// TIA Portal V20 export
// export: Created 2025-12-01T14:57:08.5701535Z, ExportSetting None, DisplayName Totally Integrated Automation Portal, DisplayVersion V20 Update 3, DisplayName TIA Portal Openness, DisplayVersion V20 Update 3, DisplayName TIA Portal Version Control Interface, DisplayVersion V20 Update 3, DisplayName STEP 7 Professional, DisplayVersion V20 Update 3, DisplayName STEP 7 Safety, DisplayVersion V20 Update 2, DisplayName WinCC Basic/Comfort/Advanced, DisplayVersion V20 Update 3, DisplayName WinCC Professional, DisplayVersion V20 Update 3, DisplayName WinCC Unified, DisplayVersion V20 Update 3
FUNCTION "FC918_GestorAccesos" : Void   // FC918, LAD
{ S7_Optimized_Access := 'FALSE' }
// stored: AutoNumber false, SetENOAutomatically false
   VAR_INPUT
      Numero : UInt;
      ModoPulsador : Bool;
      PermisoActivarPeticion : Bool;
      PermisoDesActivarPeticion : Bool;
      S_Peticion : Bool;
   END_VAR
   VAR_OUTPUT
      H_Permiso : Bool;
      NoEntrarCarga : Bool;
      BloqueoPuerta : Bool;
   END_VAR
   VAR_TEMP
      Acceso : "UDT_Accesos";
      PAny_DB_Acceso : Any;
      Guardar_AR2 : DWord;
      P_ArrayMesas : DWord;
      P_Acceso : DWord;
      ReturnValor : Int;
      Long_Accesos : UInt;
      NDB_Accesos : UInt;
      NMesas_Accesos : UInt;
      Indice : UInt;
      Mesa : UInt;
      FlancoParoBlando : Bool;
      FlancoMarcha : Bool;
      FlancoEntradaPeticion : Bool;
   END_VAR
BEGIN

NETWORK
TITLE = Inicializar
////////////////////////////////////////////////////////////////////////////////////
/// Inicializar Variables

      L     "CTE_Long_Accesos";  // Longitud de la Estructura de Accesos
      T     #Long_Accesos;
      L     "CTE_NDB_Accesos";  // Numeero DB de Accesos
      T     #NDB_Accesos;
      L     "CTE_NumMesas_Accesos";  // Numero de Mesas Max en Accesos
      T     #NMesas_Accesos;



NETWORK
TITLE = Recoger Datos del Acceso
/////////////////////////////////////////////////////////////////////////////////////
/// Puntero Any - DB de Accesos

      L     #Numero;  // Puntero al Acceso
      L     #Long_Accesos;
      *D;
      SLD   3;
      T     #P_Acceso;

      TAR2  #Guardar_AR2;
      LAR2  P##PAny_DB_Acceso;  // - Any - Datos Accesos(Temporal)
      L     B#16#10;  //   10H para S7
      T     LB [AR2, P#0.0];
      L     B#16#2;  //   Tipo de Datos (BYTE)
      T     LB [AR2, P#1.0];
      L     #Long_Accesos;  //   Cantidad de datos
      T     LW [AR2, P#2.0];
      L     #NDB_Accesos;  //   Numero de DB
      T     LW [AR2, P#4.0];
      L     #P_Acceso;  //   Direccion de Inicio
      T     LD [AR2, P#6.0];
      L     B#16#84;  //   El Area de Memoria = DB (Nota: No 84)
      T     LB [AR2, P#6.0];
      L     #Guardar_AR2;

/////////////////////////////////////////////////////////////////////////////////////
/// Cargar los Datos del Acceso

      CALL  UBLKMOV
      ( SRCBLK  := #PAny_DB_Acceso,
        RET_VAL := #ReturnValor,
        DSTBLK  := #Acceso
      );  // Copia de Datos



NETWORK
TITLE = Gestion de la Entrada de Peticion
/////////////////////////////////////////////////////////////////////////////////////
/// Seleccion del Modo

      SET;
      A     #ModoPulsador;
      JC    Activo_ModoPulsador;
      JU    Activo_ModoSelector;

/////////////////////////////////////////////////////////////////////////////////////
/// Modo Selector
Activo_ModoSelector:NOP   0;
      SET;
      A     #S_Peticion;
      =     #Acceso.Memorias.MEntradaPeticion;

      JU    Final_Modo;


/////////////////////////////////////////////////////////////////////////////////////
/// Modo Pulsador
Activo_ModoPulsador:NOP   0;
      SET;  // Control de Pulsador de la Peticion
      A     #S_Peticion;
      FP    #Acceso.Memorias.MFP_PulsadorPeticion;
      =     #FlancoEntradaPeticion;

      SET;  // Control de la Activacion del Pulsador
      AN    #Acceso.Memorias.MEntradaPeticion;
      A     #FlancoEntradaPeticion;
      JC    Activar_MPulsador_Peticion;

      SET;  // Contorl de la DesActivacion del Pulsador
      A     #Acceso.Memorias.MEntradaPeticion;
      A     #FlancoEntradaPeticion;
      JC    DesActivar_MPulsador_Peticion;

      JU    Final_Modo;  // No se ha pulsado


/// Activar Memoria del Pulsador de Peticion
Activar_MPulsador_Peticion:NOP   0;
      SET;
      S     #Acceso.Memorias.MEntradaPeticion;
      JU    Final_Modo;


/// DesActivar Memoria del Pulsador de Peticion
DesActivar_MPulsador_Peticion:NOP   0;
      SET;
      R     #Acceso.Memorias.MEntradaPeticion;
      JU    Final_Modo;


/////////////////////////////////////////////////////////////////////////////////////
/// Final de la Seleccion del Modo
Final_Modo:NOP   0;


NETWORK
TITLE = Gestion de Peticion
/////////////////////////////////////////////////////////////////////////////////////
/// Gestion de la Peticion de Acceso

      SET;  // Activacion de la Peticion
      A     #Acceso.Memorias.MEntradaPeticion;
      A     #PermisoActivarPeticion;
      S     #Acceso.Memorias.MPeticion;

      SET;  // DesActivacion de la Peticion
      AN    #Acceso.Memorias.MEntradaPeticion;
      A     #PermisoDesActivarPeticion;
      R     #Acceso.Memorias.MPeticion;



NETWORK
TITLE = Estado de las Mesas existentes en el Acceso
/////////////////////////////////////////////////////////////////////////////////////
/// Todas las Mesas estan en Paro

      SET;
      S     #Acceso.Memorias.TodasMesas_EnParo;
      R     #Acceso.Memorias.AlgunaMesa_EnMarcha;

      L     P##Acceso;  // Puntero al Array de Mesas
      L     P#2.0;
      +D;
      T     #P_ArrayMesas;

      L     #NMesas_Accesos;  // Bucle de Numero Total de Mesas existentes
BucleMesas:NOP   0;
      T     #Indice;

      L     LW [#P_ArrayMesas];
      T     #Mesa;

      L     0;  // Existe Mesa
      L     #Mesa;
      ==I;
      JC    FinBucleMesas;


      SET;
      A     "DB902_Estado_ZonaMesa".EstadoMesas[#Mesa].Marcha_CBx;
      R     #Acceso.Memorias.TodasMesas_EnParo;

      SET;
      A     #Acceso.Memorias.AlgunaMesa_EnMarcha;
      O     "DB902_Estado_ZonaMesa".EstadoMesas[#Mesa].Marcha_CBx;
      S     #Acceso.Memorias.AlgunaMesa_EnMarcha;

      L     #P_ArrayMesas;  // Siguiente Mesa
      L     P#2.0;
      +D;
      T     #P_ArrayMesas;

      L     #Indice;
      LOOP  BucleMesas;  //  Final del Testeo


/////////////////////////////////////////////////////////////////////////////////////
/// Final
FinBucleMesas:NOP   0;



NETWORK
TITLE = Gestion de Permiso
/////////////////////////////////////////////////////////////////////////////////////
/// Gestion del Permiso de Acceso

      SET;  // Activacion del Permiso
      A     #Acceso.Memorias.TodasMesas_EnParo;
      A     #Acceso.Memorias.MPeticion;
      S     #Acceso.Memorias.MPermiso;

      SET;  // DesActivacion del Permiso
      AN    #Acceso.Memorias.MPeticion;
      R     #Acceso.Memorias.MPermiso;



NETWORK
TITLE = Gestion de Paro Blando
/////////////////////////////////////////////////////////////////////////////////////
/// Gestion de Paro Blando

      A     #Acceso.Memorias.MPeticion;
      A     #Acceso.Memorias.AlgunaMesa_EnMarcha;
      FP    #Acceso.Memorias.MFP_ParoBlando;
      =     #FlancoParoBlando;


/////////////////////////////////////////////////////////////////////////////////////
/// Activacion del Paro Blando

      SET;
      AN    #FlancoParoBlando;
      JC    FinParoBlandoMesas;

      L     P##Acceso;  // Puntero al Array de Mesas
      L     P#2.0;
      +D;
      T     #P_ArrayMesas;

      L     #NMesas_Accesos;  // Bucle de Numero Total de Mesas existentes
BucleMesas_ParoBlando:T     #Indice;

      L     LW [#P_ArrayMesas];
      T     #Mesa;

      L     0;  // Existe Mesa
      L     #Mesa;
      ==I;
      JC    FinParoBlandoMesas;

      SET;  // Activar La Orden de Paro Blando de la Mesa
      S     "DB843_RecepcionPantalla".Mesa[#Mesa].ParoBlando;

      L     #P_ArrayMesas;  // Siguiente Mesa
      L     P#2.0;
      +D;
      T     #P_ArrayMesas;

      L     #Indice;
      LOOP  BucleMesas_ParoBlando;  //  Final del Testeo


/////////////////////////////////////////////////////////////////////////////////////
/// Final del Paro Blando
FinParoBlandoMesas:NOP   0;



NETWORK
TITLE = Gestion de Marcha
/////////////////////////////////////////////////////////////////////////////////////
/// Gestion de la Marcha

      AN    #Acceso.Memorias.MPeticion;
      FP    #Acceso.Memorias.MFP_Marcha;
      =     #FlancoMarcha;


/////////////////////////////////////////////////////////////////////////////////////
/// Activacion de la Marcha

      SET;
      AN    #FlancoMarcha;
      JC    FinMarchaMesas;

      L     P##Acceso;  // Puntero al Array de Mesas
      L     P#2.0;
      +D;
      T     #P_ArrayMesas;

      L     #NMesas_Accesos;  // Bucle de Numero Total de Mesas existentes
BucleMesas_Marcha:T     #Indice;

      L     LW [#P_ArrayMesas];
      T     #Mesa;

      L     0;  // Existe Mesa
      L     #Mesa;
      ==I;
      JC    FinMarchaMesas;

      SET;  // Activar La Orden de Marcha de la Mesa
      S     "DB843_RecepcionPantalla".Mesa[#Mesa].Marcha;

      L     #P_ArrayMesas;  // Siguiente Mesa
      L     P#2.0;
      +D;
      T     #P_ArrayMesas;

      L     #Indice;
      LOOP  BucleMesas_Marcha;  //  Final del Testeo


/////////////////////////////////////////////////////////////////////////////////////
/// Final de la Marcha
FinMarchaMesas:NOP   0;



NETWORK
TITLE = Final de la Funcion
/////////////////////////////////////////////////////////////////////////////////////
/// Guardar los Datos del Acceso

      CALL  UBLKMOV
      ( SRCBLK  := #Acceso,
        RET_VAL := #ReturnValor,
        DSTBLK  := #PAny_DB_Acceso
      );  // Copia de Datos



REGION Network 10: Activacion de Salidas del Acceso
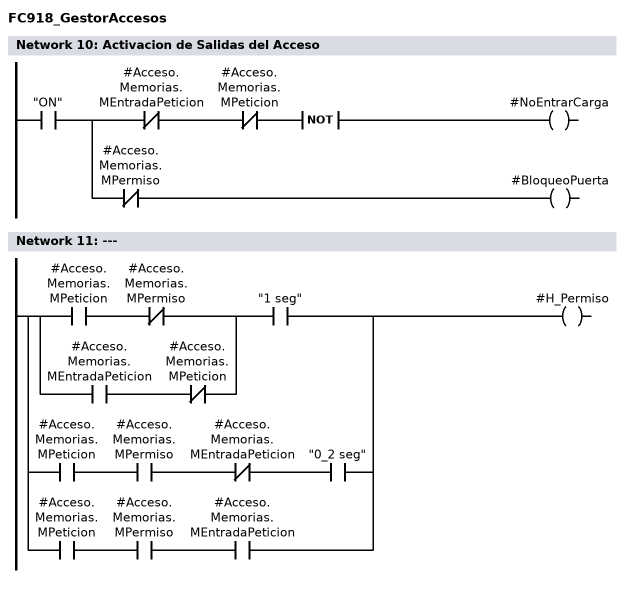
   RUNG wire#powerrail
      Contact( "ON" )
      wire#w1
      I_Contact( #Acceso.Memorias.MEntradaPeticion )
      I_Contact( #Acceso.Memorias.MPeticion )
      Not()
      Coil( #NoEntrarCarga )
   END_RUNG
   RUNG wire#w1
      I_Contact( #Acceso.Memorias.MPermiso )
      Coil( #BloqueoPuerta )
   END_RUNG
   // the same network as SCL:
   #NoEntrarCarga := NOT ("ON" AND NOT #Acceso.Memorias.MEntradaPeticion AND NOT #Acceso.Memorias.MPeticion);
   #BloqueoPuerta := "ON" AND NOT #Acceso.Memorias.MPermiso;
END_REGION

REGION Network 11: ---
   RUNG wire#powerrail
      Contact( #Acceso.Memorias.MPeticion )
      I_Contact( #Acceso.Memorias.MPermiso )
      wire#w1
      Contact( "1 seg" )
      wire#w2
      Coil( #H_Permiso )
   END_RUNG
   RUNG wire#powerrail
      Contact( #Acceso.Memorias.MEntradaPeticion )
      I_Contact( #Acceso.Memorias.MPeticion )
   END_RUNG wire#w1
   RUNG wire#powerrail
      Contact( #Acceso.Memorias.MPeticion )
      Contact( #Acceso.Memorias.MPermiso )
      I_Contact( #Acceso.Memorias.MEntradaPeticion )
      Contact( "0_2 seg" )
   END_RUNG wire#w2
   RUNG wire#powerrail
      Contact( #Acceso.Memorias.MPeticion )
      Contact( #Acceso.Memorias.MPermiso )
      Contact( #Acceso.Memorias.MEntradaPeticion )
   END_RUNG wire#w2
   // the same network as SCL:
   #H_Permiso := (((#Acceso.Memorias.MPeticion AND NOT #Acceso.Memorias.MPermiso) OR (#Acceso.Memorias.MEntradaPeticion AND NOT #Acceso.Memorias.MPeticion)) AND "1 seg") OR (#Acceso.Memorias.MPeticion AND #Acceso.Memorias.MPermiso AND NOT #Acceso.Memorias.MEntradaPeticion AND "0_2 seg") OR (#Acceso.Memorias.MPeticion AND #Acceso.Memorias.MPermiso AND #Acceso.Memorias.MEntradaPeticion);
END_REGION

REGION Network 12: ---
END_REGION
END_FUNCTION
